(* CoDeSys 2.3.9.62 project: Cap6_ej1.pro *)
(* Libraries: Standard.lib 4.10.05 11:14:46, IecSfc.lib*2.6.14 10:37:46 *)

(* POU PLC_PRG, LD *)
PROGRAM PLC_PRG
VAR
   (* Entradas *)
	A: BOOL;
       B:BOOL;
	C: BOOL;

   (*Salidas *)
	S1: BOOL;
	S2: BOOL;
	S3: BOOL;
	S4: BOOL;
END_VAR
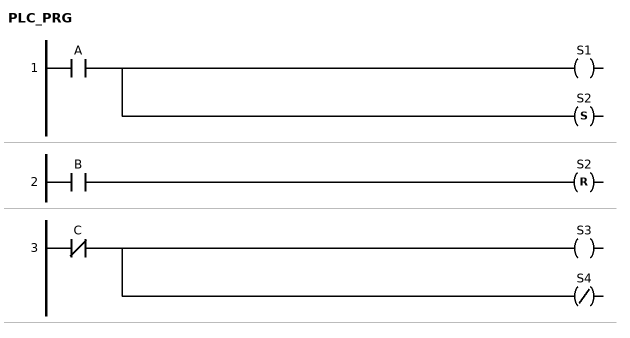
_LD_ (* Ladder Diagram *)
NETWORK 1
	[A] --- (S1) (S S2)
NETWORK 2
	[B] --- (R S2)
NETWORK 3
	[/C] --- (S3) (/S4)
_END_LD_
(* the same logic as Structured Text *)
(* Network 1 *)
S1 := A;
IF A THEN S2 := TRUE; END_IF;
(* Network 2 *)
IF B THEN S2 := FALSE; END_IF;
(* Network 3 *)
S3 := NOT C;
S4 := NOT S3;
END_PROGRAM

(* Visualisation Visu
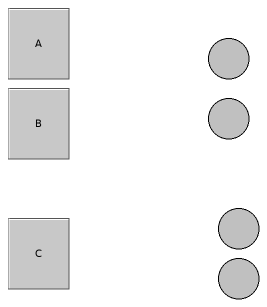
button at (60,40)-(121,111): text "A"; taps PLC_PRG.A
ellipse at (260,70)-(301,111): alarm colour if PLC_PRG.S1
ellipse at (260,130)-(301,171): alarm colour if PLC_PRG.S2
button at (60,120)-(121,191): text "B"; taps PLC_PRG.B
button at (60,250)-(121,321): text "C"; toggles PLC_PRG.C
ellipse at (270,240)-(311,281): alarm colour if PLC_PRG.S3
ellipse at (270,290)-(311,331): alarm colour if PLC_PRG.S4
6 elements of other kinds (tables, trends, ...) not read
*)
